FUNCTION F_GetDorPressure : real
VAR_INPUT
	nPressurePV:INT;
END_VAR

VAR
	Value:REAL;
END_VAR

Value:= (10.0 / 32767.0) * nPressurePV;
F_GetDorPressure := (190* (Value) ) - 190;

END_FUNCTION

(* stored: Version 1.1.0.1, ProductVersion 3.1.4024.15
   POU F_GetDorPressure: Id {d5eb6636-a4af-417e-be51-f91c045e6ee3}, SpecialFunc None *)
